Fanuc TP program (LS listing): MON_OKUMA2.LS

/PROG  MON_OKUMA2	  Cond
/ATTR
OWNER		= MNEDITOR;
COMMENT		= "MONITOR MACHINE";
PROG_SIZE	= 239;
CREATE		= DATE 20-02-05  TIME 02:01:40;
MODIFIED	= DATE 20-02-05  TIME 02:02:08;
FILE_NAME	= MON_OP20;
VERSION		= 0;
LINE_COUNT	= 1;
MEMORY_SIZE	= 615;
PROTECT		= READ_WRITE;
TCD:  STACK_SIZE	= 0,
      TASK_PRIORITY	= 50,
      TIME_SLICE	= 0,
      BUSY_LAMP_OFF	= 0,
      ABORT_REQUEST	= 0,
      PAUSE_REQUEST	= 0;
DEFAULT_GROUP	= *,*,*,*,*;
CONTROL_CODE	= 00000000 00000000;
/APPL

AUTO_SINGULARITY_HEADER;
  ENABLE_SINGULARITY_AVOIDANCE   : TRUE;
/MN
   1:  WHEN DO[124:OFF:OK2 SAFE FOR ROBOT]=OFF,CALL MON_OP20_1ALM ;
/POS
/END
